# EPICS substitutions: modules/event/evrSupport/Db/ioc/IOC-LI21-PM01evr.substitutions
#==============================================================================
#
# Abs:  LCLS EVR IOC records for LI21 PM01
#
# Name: IOC-LI21-PM01evr.substitutions
#
#==============================================================================
#
file evrPMXX.db
{
pattern { DEVICE        }
	{ EVR:LI21:PM01 }
}
